TYPE stAi4CH :
STRUCT
	CH1 AT %I* : INT;
	CH2 AT %I* : INT;
	CH3 AT %I* : INT;
	CH4 AT %I* : INT;
END_STRUCT
END_TYPE

(* stored: Version 1.1.0.1, ProductVersion 3.1.4024.2
   DUT stAi4CH: Id {b25bbdb0-7f56-4704-85b1-09d56ef3dbf6} *)
